// TIA Portal V20 export
DATA_BLOCK "LBP_TMLoadMT"   // DB1071
TITLE = Tool management / Gestion des outils
{ S7_Optimized_Access := 'FALSE' }
AUTHOR : SINUMERIK
FAMILY : SINUMERIK_ONE
VERSION : 6.24
// Interface between user program and tool management, contains signals from/to Load/Unload magazine (multitool). / Interface entre programme utilisateur et gestion d'outil, contient des signaux de/vers Chargement/déchargement de magasin (Multitool).
// stored: AutoNumber false, InstanceOfName LBP_typeTMLoadMT, InstanceOfType UDT
"LBP_typeTMLoadMT"
   // VAR RETAIN
   //    MTIF : Array[1..16] of Struct
   //       DistanceCoding : Int;
   //       Places : Int;
   //       Distance : Real;
   //       MTNo : Int;
   //       PlaceNo : Int;
   //       Toolholder : Int;
   //       reserved : Array[1..3] of Int;
   //    END_STRUCT;
   // END_VAR
BEGIN
END_DATA_BLOCK
